// TwinCAT 3 PLC project PLC1
// ProgramVersion: 3.1.4023.0
// libraries:
//   Tc2_Standard, * (Beckhoff Automation GmbH)
//   Tc2_System, * (Beckhoff Automation GmbH)
//   Tc3_Module, * (Beckhoff Automation GmbH)
// project tree:
//   / GlobalTextList.TcGTLO (not stored), PlcTask.TcTTO (not stored)
//   GVLs/ Devices.TcGVL (not stored), GVL.TcGVL
//   POUs/Devices/ FB_MotorContactor.TcPOU (not stored), FB_NormallyClosedPB.TcPOU, FB_NormallyClosedSensor.TcPOU, FB_NormallyOpenPB.TcPOU (not stored), FB_NormallyOpenSensor.TcPOU (not stored)
//   POUs/ I_Pushbutton.TcIO (not stored), I_Sensor.TcIO (not stored), MAIN.TcPOU (not stored)
//   POUs/Machine/ FB_ConveyorMachine.TcPOU
// real-time tasks:
//   TASK PlcTask: cycle T#10ms, priority 20, ADS port 350

// ---- GVLs/GVL.TcGVL
{attribute 'qualified_only'}
VAR_GLOBAL
	StopButton 					AT %I* : BOOL;
	EmergencyStopButton 		AT %I* : BOOL;
	StartButton 				AT %I* : BOOL;
	ProductDetectedSensor 		AT %I* : BOOL;
	ConveyorFullSensor 			AT %I* : BOOL;
	MotorContactor 				AT %Q* : BOOL;
END_VAR

// ---- POUs/Devices/FB_NormallyClosedPB.TcPOU
FUNCTION_BLOCK FB_NormallyClosedPB IMPLEMENTS I_Pushbutton
VAR
	Input AT %I* : BOOL;
END_VAR

PROPERTY IsPressed : BOOL
GET
IsPressed := NOT Input;
END_GET
END_PROPERTY

PROPERTY IsReleased : BOOL
GET
IsReleased := Input;
END_GET
END_PROPERTY

END_FUNCTION_BLOCK

// ---- POUs/Devices/FB_NormallyClosedSensor.TcPOU
FUNCTION_BLOCK FB_NormallyClosedSensor IMPLEMENTS I_Sensor
VAR
	Input AT %I* : BOOL;
END_VAR

{warning 'add property implementation'}
PROPERTY IsActive : BOOL
GET
IsActive := NOT Input;
END_GET
END_PROPERTY

END_FUNCTION_BLOCK

// ---- POUs/Machine/FB_ConveyorMachine.TcPOU
FUNCTION_BLOCK FB_ConveyorMachine
VAR
	StopButton 				: I_Pushbutton;
	EmergencyStopButton 	: I_Pushbutton;
	StartButton 			: I_Pushbutton;
	ProductDetectedSensor 	: I_Sensor;
	ConveyorFullSensor		: I_Sensor;
	MotorContactor 			: FB_MotorContactor;
	Timeout 				: TOF;
	ConveyorControl 		: BOOL;
END_VAR

IF StopButton.IsPressed OR EmergencyStopButton.IsPressed THEN	
	ConveyorControl := FALSE;	
ELSIF StartButton.IsPressed AND StopButton.IsReleased AND EmergencyStopButton.IsReleased THEN
	ConveyorControl := TRUE;	
END_IF

Timeout(IN:= ConveyorControl AND ProductDetectedSensor.IsActive, PT:= T#5S);

IF ConveyorControl AND Timeout.Q AND NOT ConveyorFullSensor.IsActive THEN
	MotorContactor.SwitchOn();
ELSE
	MotorContactor.SwitchOff();
END_IF

METHOD FB_init : BOOL
VAR_INPUT
	bInitRetains : BOOL; // if TRUE, the retain variables are initialized (warm start / cold start)
	bInCopyCode : BOOL;  // if TRUE, the instance afterwards gets moved into the copy code (online change)
	StopButton 				: I_Pushbutton;
	EmergencyStopButton 	: I_Pushbutton;
	StartButton 			: I_Pushbutton;
	ProductDetectedSensor 	: I_Sensor;
	ConveyorFullSensor		: I_Sensor;
	MotorContactor 			: FB_MotorContactor;
END_VAR
THIS^.StopButton 				:= StopButton 			;	        
THIS^.EmergencyStopButton 		:= EmergencyStopButton 	;  
THIS^.StartButton 				:= StartButton 			;        
THIS^.ProductDetectedSensor 	:= ProductDetectedSensor; 	
THIS^.ConveyorFullSensor		:= ConveyorFullSensor	;	   
THIS^.MotorContactor 			:= MotorContactor 		;
END_METHOD

END_FUNCTION_BLOCK
